// Mitsubishi GX Works2 project: PLC_GROUP21   PLC: FX3G

// global labels: Global1
VAR_GLOBAL
  start_day_switch AT X007 : BOOL;
  start_day_light AT Y007 : BOOL;
  end_day_light AT M3 : BOOL;
  input1 AT D1110 : REAL;
  input2 AT D1120 : REAL;
  input3 AT D1130 : REAL;
  input4 AT D1140 : REAL;
  petel AT D1150 : REAL;
  lemon AT D1160 : REAL;
  stabilizer AT D1170 : REAL;
  gummybears AT D1180 : REAL;
  prepare_switch AT X001 : BOOL;
  regular_gumigam_range AT M20 : BOOL;
  deluxe_gumigam_range AT M19 : BOOL;
END_VAR
VAR_GLOBAL CONSTANT
  const5 : REAL := 5.0;
  const6 : REAL := 6.0;
  divide : REAL := 400.0;
END_VAR
VAR_GLOBAL
  saved_analog AT D7000 : REAL;
  analog_input1 AT D8280 : INT;
END_VAR
VAR_GLOBAL CONSTANT
  min_pete_regular : REAL := 280;
END_VAR
VAR_GLOBAL
  enough_petel_regular AT M60 : BOOL;
END_VAR
VAR_GLOBAL CONSTANT
  min_lemon_regular : REAL := 455;
END_VAR
VAR_GLOBAL
  enough_lemon_regular AT M61 : BOOL;
END_VAR
VAR_GLOBAL CONSTANT
  min_stabilizer_regular : REAL := 105;
END_VAR
VAR_GLOBAL
  enough_gumi_bears AT M63 : BOOL;
END_VAR
VAR_GLOBAL CONSTANT
  min_gummybears_regular : REAL := 28;
END_VAR
VAR_GLOBAL
  enough_stabilizer_regular AT M62 : BOOL;
END_VAR
VAR_GLOBAL CONSTANT
  min_pete_del : REAL := 385;
END_VAR
VAR_GLOBAL
  enough_petel_del AT M50 : BOOL;
END_VAR
VAR_GLOBAL CONSTANT
  min_lemon_del : REAL := 665;
END_VAR
VAR_GLOBAL
  enough_lemon_del AT M51 : BOOL;
END_VAR
VAR_GLOBAL CONSTANT
  min_stabilizer_del : REAL := 210;
END_VAR
VAR_GLOBAL
  enough_stabilizer_del AT M52 : BOOL;
END_VAR
VAR_GLOBAL CONSTANT
  min_gummybears_del : REAL := 70;
END_VAR
VAR_GLOBAL
  enough_gummybears_regular AT M63 : BOOL;
  enough_gummybears_del AT M53 : BOOL;
  help_gate_regular AT M39 : BOOL;
  help_gate_del AT M38 : BOOL;
  enough_in_regularl_stock AT M18 : BOOL;
  enough_in_del_stock AT M40 : BOOL;
  preper_icecream_timer AT TC9 : BOOL;
  const_5 AT K50 : INT;
  preper_icecream_timer_ts9 AT TS9 : BOOL;
  preper_icecream_is_on_light AT Y000 : BOOL;
  preper_is_on_light AT Y000 : BOOL;
END_VAR
VAR_GLOBAL CONSTANT
  time_for_cold_8S : INT := 80;
END_VAR
VAR_GLOBAL
  time_fer AT D1180 : INT;
  sen_10 AT X003 : BOOL;
END_VAR
VAR_GLOBAL CONSTANT
  time_for_fer_const_3S : INT := 3;
  time_for_mix_5S : INT := 50;
  time_for_mix_3S : INT := 30;
END_VAR
VAR_GLOBAL
  Y5_light_on AT Y005 : BOOL;
  Y6_light_on AT Y006 : BOOL;
  Y6_flash_counter AT TC6 : BOOL;
  timer_ts6 AT TS6 : BOOL;
  finish_cold : BOOL;
  packing_switch AT X004 : BOOL;
  counter_pack AT CC3 : BOOL;
  Y4_light_on AT Y004 : BOOL;
  CC3_term AT CS3 : BOOL;
END_VAR
VAR_GLOBAL CONSTANT
  const7 : INT := 7;
  pack_finish : REAL := 1.0;
END_VAR
VAR_GLOBAL
  cont_petel_ice_cream AT D1190 : REAL;
  cont_lemon_ice_cream AT D1200 : REAL;
END_VAR
VAR_GLOBAL CONSTANT
  lemon_for_petel_icecream_regular : REAL := 35;
  stabilizer_for_petel_ice_regular : REAL := 35;
  stabilizer_for_del_icecream : REAL := 140;
  lemon_for_del_icecream : REAL := 560;
  lemon_for_del_lemon_icecream : REAL := 560;
  lemon_for_lemon_icecream_regular : REAL := 420;
  stabilizer_for_lemon_ice_regular : REAL := 70;
  lemon_for_petel_icecream_del : REAL := 105;
  stabilizer_for_petel_ice_del : REAL := 70;
END_VAR
VAR_GLOBAL
  start_cooling AT X002 : BOOL;
  cooling_petel AT D1300 : REAL;
  cooling_lemon AT D1310 : REAL;
END_VAR
VAR_GLOBAL CONSTANT
  stabilizer_for_del_lemon_ice : REAL := 140;
END_VAR
VAR_GLOBAL
  cooling_icecream_timer AT TC8 : BOOL;
  const_8 AT K80 : INT;
  cooling_icecream_timer_ts8 AT TS8 : BOOL;
  cooling_icecream_is_on_light AT Y002 : BOOL;
  stop_cooling AT M10 : BOOL;
END_VAR
VAR_GLOBAL CONSTANT
  update_petel_cont : REAL := 350;
  update_reg_lemon_cont : REAL := 490;
  update_reg_petel_cont : REAL := 350;
  update_del_petel_cont : REAL := 560;
  update_del_lemon_cont : REAL := 700;
END_VAR
VAR_GLOBAL
  mix_cont AT D1320 : REAL;
  time_mix AT D1500 : INT;
  mix_flash_counter AT TC4 : BOOL;
  mix_flash_counter_ts4 AT TS4 : BOOL;
  const_1 AT K10 : INT;
  mix_time_reg AT TC3 : BOOL;
  mix_time_del AT TC5 : BOOL;
END_VAR
VAR_GLOBAL CONSTANT
  const_time_mix_reg : INT := 30;
  const_time_mix_del : INT := 50;
END_VAR
VAR_GLOBAL
  mix_time_reg_ts AT TS3 : BOOL;
  mix_time_del_ts AT TS5 : BOOL;
  start_blinking AT M36 : BOOL;
  Y5_flash_counter AT TC7 : BOOL;
  timer_ts7 AT TS7 : BOOL;
  blink_time AT K10 : INT;
  blinking_help AT M37 : BOOL;
  pack1_switch AT X000 : BOOL;
  count_gumigam_in_box AT CN3 : INT;
END_VAR
VAR_GLOBAL CONSTANT
  no_gumigam : INT;
END_VAR
VAR_GLOBAL
  new_box AT M70 : BOOL;
  end_day_switch AT X005 : BOOL;
  analog_output AT D8282 : INT;
END_VAR
VAR_GLOBAL CONSTANT
  const_40 : REAL := 40;
END_VAR
VAR_GLOBAL
  reg_pack_count_after_mul AT D1404 : REAL;
  input1_petel AT D1110 : REAL;
  input2_lemon AT D1120 : REAL;
  input3_stabilizer AT D1130 : REAL;
  input4_gummybears AT D1140 : REAL;
  pack_total_count AT D1402 : REAL;
  zero AT D5000 : REAL;
  zero_word AT D5010 : INT;
  cont AT D1200 : REAL;
  end_of_iteration AT M80 : BOOL;
  bDIKA AT M90 : BOOL;
END_VAR

// task Task_01 (event TRUE, interval 0, priority 31): POU_01

PROGRAM POU_01
(* structured ladder/FBD written out as ST: instructions are called as NAME(EN, inputs, outputs); _pN, _eN, _tN stand for wires *)
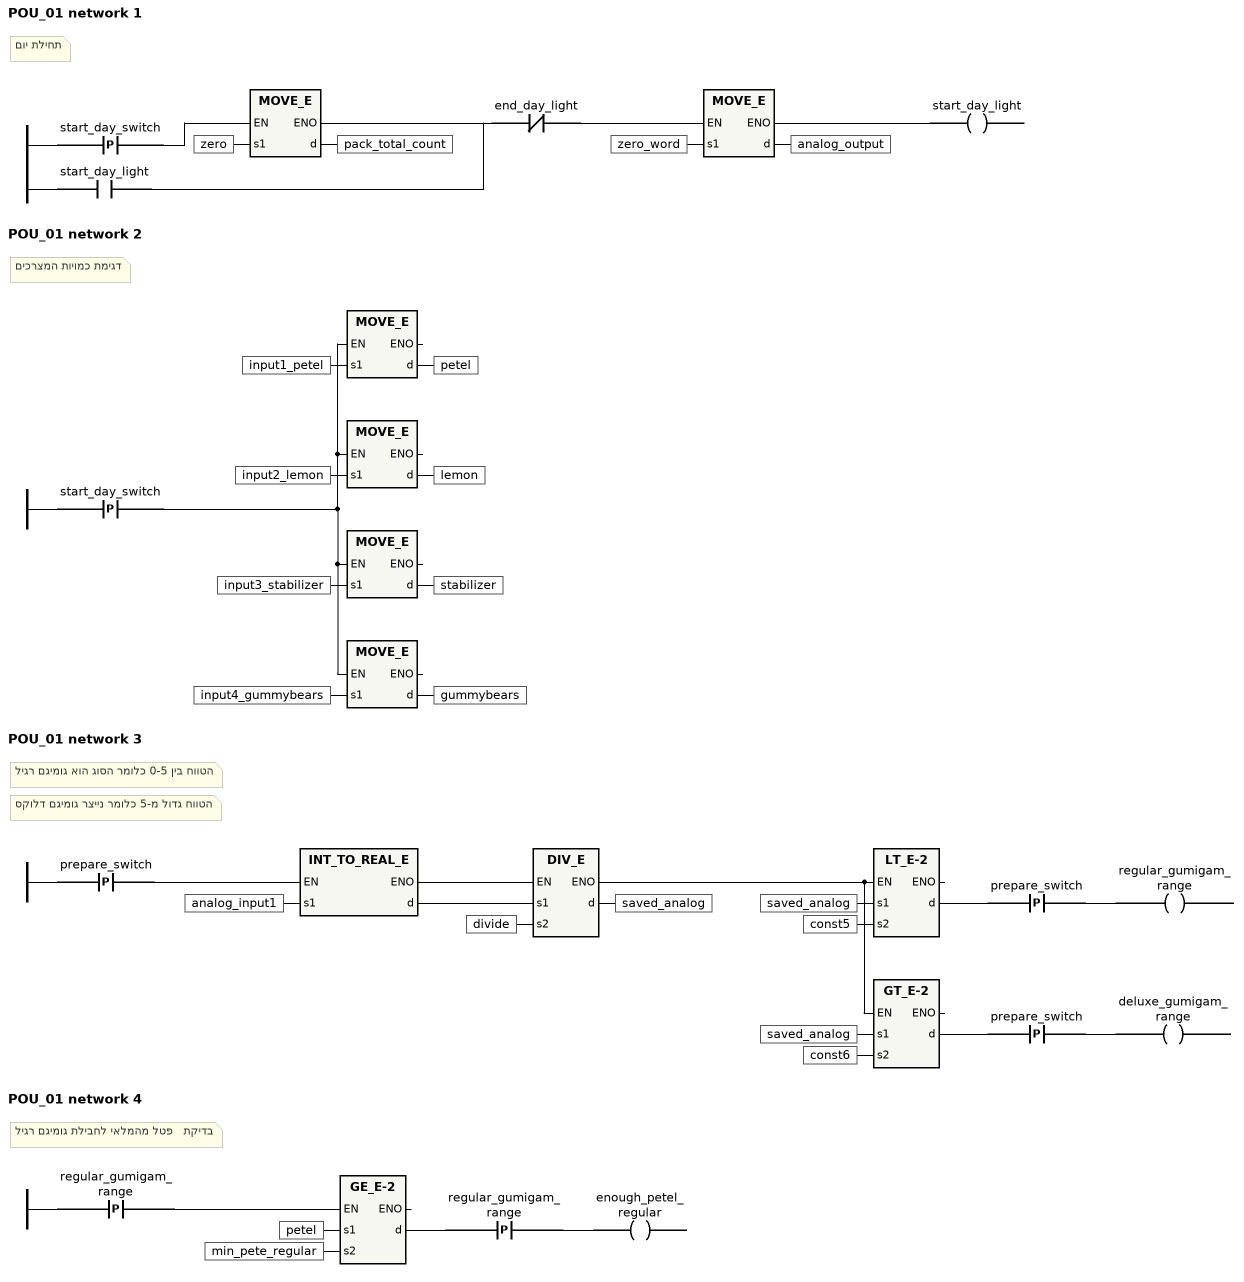
(* network 1 *)
(* תחילת יום *)
_e1 := MOVE_E(LDP(TRUE, start_day_switch), zero, pack_total_count);
_e2 := MOVE_E((_e1 OR start_day_light) AND NOT end_day_light, zero_word, analog_output);
start_day_light := _e2;
(* network 2 *)
(* דגימת כמויות המצרכים *)
_p1 := LDP(TRUE, start_day_switch);
MOVE_E(_p1, input1_petel, petel);
MOVE_E(_p1, input2_lemon, lemon);
MOVE_E(_p1, input3_stabilizer, stabilizer);
MOVE_E(_p1, input4_gummybears, gummybears);
(* network 3 *)
(* הטווח בין 0-5 כלומר הסוג הוא גומיגם רגיל *)
(* הטווח גדול מ-5 כלומר נייצר גומיגם דלוקס *)
_e2 := INT_TO_REAL_E(LDP(TRUE, prepare_switch), analog_input1, _t1);
_e3 := DIV_E(_e2, _t1, divide, saved_analog);
LT_E(_e3, saved_analog, const5, _t4);
regular_gumigam_range := _t4 AND LDP(TRUE, prepare_switch);
GT_E(_e3, saved_analog, const6, _t5);
deluxe_gumigam_range := _t5 AND LDP(TRUE, prepare_switch);
(* network 4 *)
(* בדיקת   פטל מהמלאי לחבילת גומיגם רגיל *)
GE_E(LDP(TRUE, regular_gumigam_range), petel, min_pete_regular, _t1);
enough_petel_regular := _t1 AND LDP(TRUE, regular_gumigam_range);
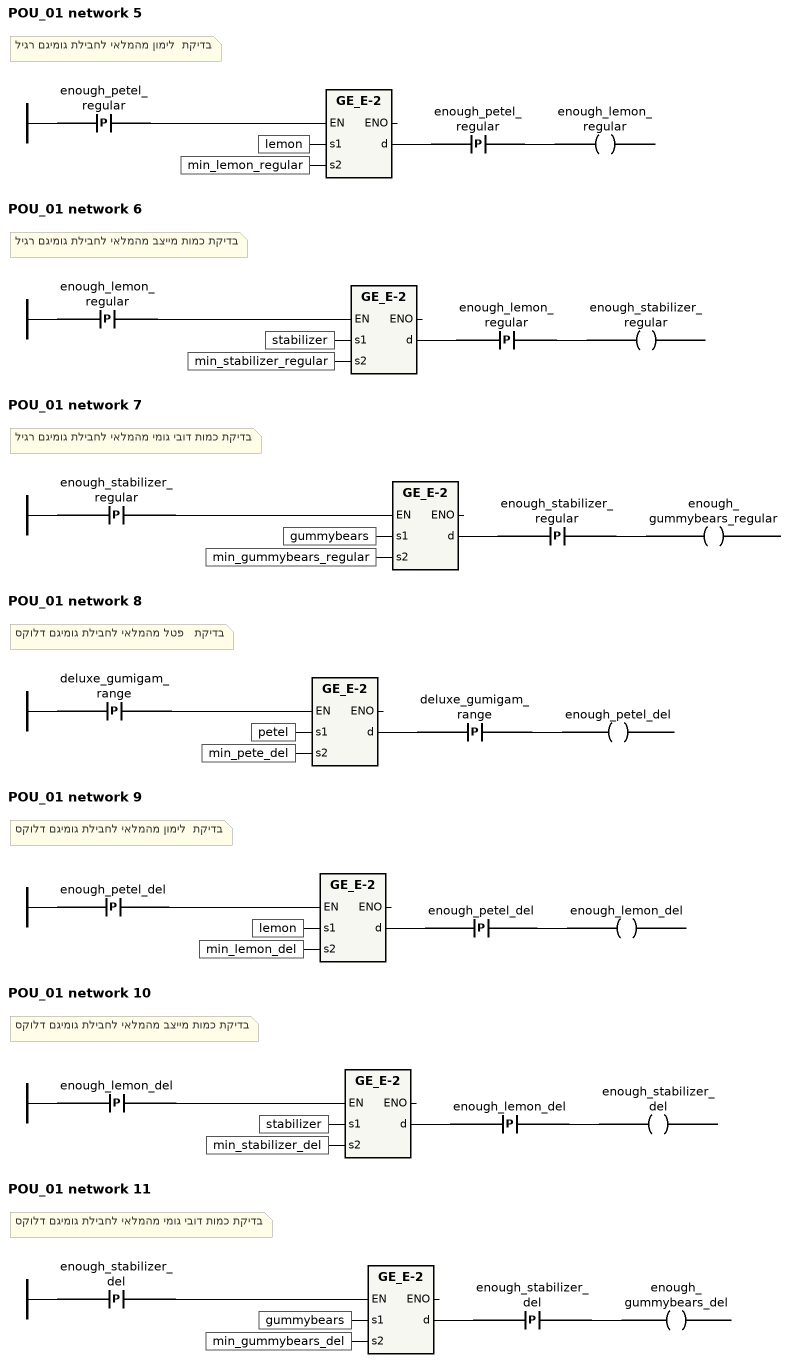
(* network 5 *)
(* בדיקת  לימון מהמלאי לחבילת גומיגם רגיל *)
GE_E(LDP(TRUE, enough_petel_regular), lemon, min_lemon_regular, _t1);
enough_lemon_regular := _t1 AND LDP(TRUE, enough_petel_regular);
(* network 6 *)
(* בדיקת כמות מייצב מהמלאי לחבילת גומיגם רגיל *)
GE_E(LDP(TRUE, enough_lemon_regular), stabilizer, min_stabilizer_regular, _t1);
enough_stabilizer_regular := _t1 AND LDP(TRUE, enough_lemon_regular);
(* network 7 *)
(* בדיקת כמות דובי גומי מהמלאי לחבילת גומיגם רגיל *)
GE_E(LDP(TRUE, enough_stabilizer_regular), gummybears, min_gummybears_regular, _t1);
enough_gummybears_regular := _t1 AND LDP(TRUE, enough_stabilizer_regular);
(* network 8 *)
(* בדיקת   פטל מהמלאי לחבילת גומיגם דלוקס *)
GE_E(LDP(TRUE, deluxe_gumigam_range), petel, min_pete_del, _t1);
enough_petel_del := _t1 AND LDP(TRUE, deluxe_gumigam_range);
(* network 9 *)
(* בדיקת  לימון מהמלאי לחבילת גומיגם דלוקס *)
GE_E(LDP(TRUE, enough_petel_del), lemon, min_lemon_del, _t1);
enough_lemon_del := _t1 AND LDP(TRUE, enough_petel_del);
(* network 10 *)
(* בדיקת כמות מייצב מהמלאי לחבילת גומיגם דלוקס *)
GE_E(LDP(TRUE, enough_lemon_del), stabilizer, min_stabilizer_del, _t1);
enough_stabilizer_del := _t1 AND LDP(TRUE, enough_lemon_del);
(* network 11 *)
(* בדיקת כמות דובי גומי מהמלאי לחבילת גומיגם דלוקס *)
GE_E(LDP(TRUE, enough_stabilizer_del), gummybears, min_gummybears_del, _t1);
enough_gummybears_del := _t1 AND LDP(TRUE, enough_stabilizer_del);
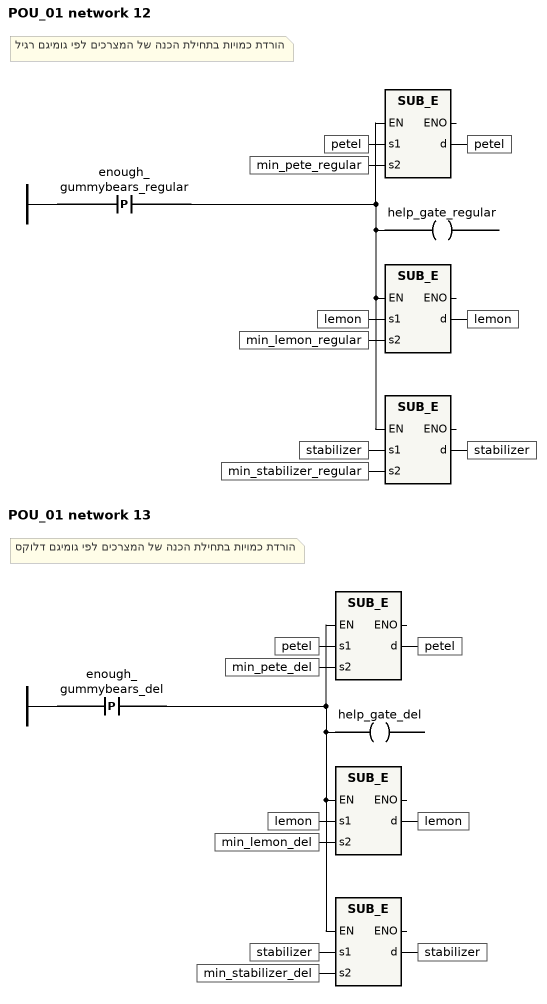
(* network 12 *)
(* הורדת כמויות בתחילת הכנה של המצרכים לפי גומיגם רגיל *)
_p1 := LDP(TRUE, enough_gummybears_regular);
help_gate_regular := _p1;
SUB_E(_p1, petel, min_pete_regular, petel);
SUB_E(_p1, lemon, min_lemon_regular, lemon);
SUB_E(_p1, stabilizer, min_stabilizer_regular, stabilizer);
(* network 13 *)
(* הורדת כמויות בתחילת הכנה של המצרכים לפי גומיגם דלוקס *)
_p1 := LDP(TRUE, enough_gummybears_del);
help_gate_del := _p1;
SUB_E(_p1, petel, min_pete_del, petel);
SUB_E(_p1, lemon, min_lemon_del, lemon);
SUB_E(_p1, stabilizer, min_stabilizer_del, stabilizer);
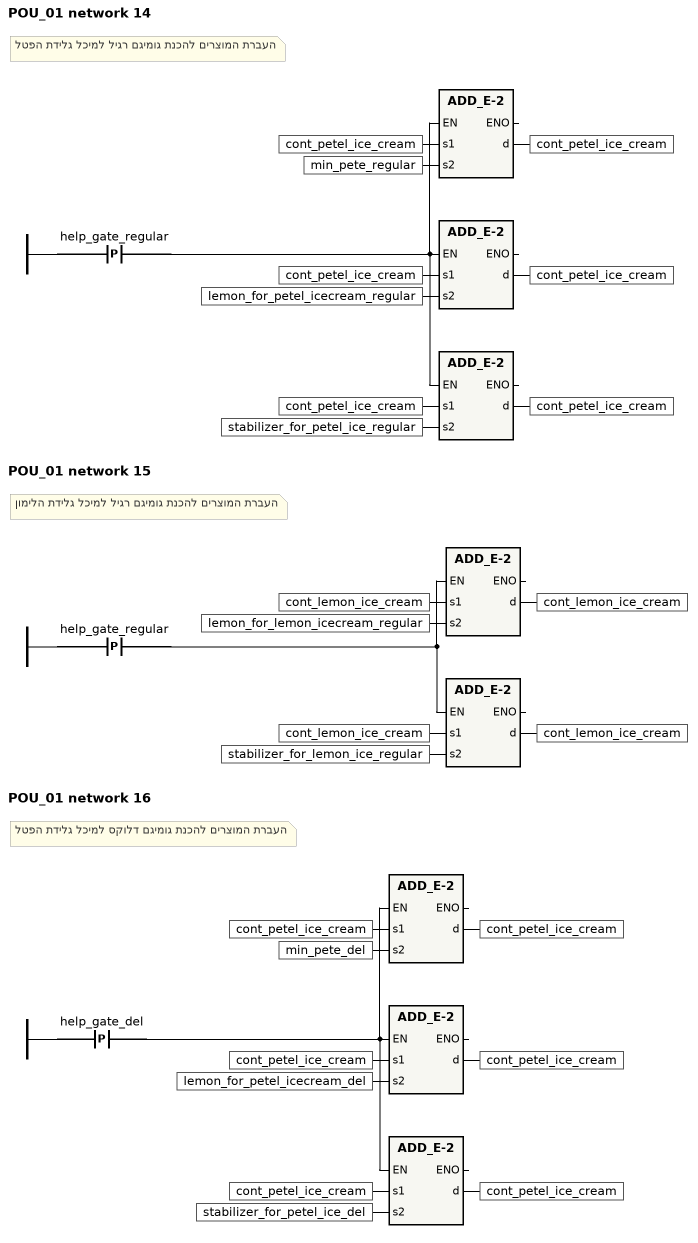
(* network 14 *)
(* העברת המוצרים להכנת גומיגם רגיל למיכל גלידת הפטל *)
_p1 := LDP(TRUE, help_gate_regular);
ADD_E(_p1, cont_petel_ice_cream, min_pete_regular, cont_petel_ice_cream);
ADD_E(_p1, cont_petel_ice_cream, lemon_for_petel_icecream_regular, cont_petel_ice_cream);
ADD_E(_p1, cont_petel_ice_cream, stabilizer_for_petel_ice_regular, cont_petel_ice_cream);
(* network 15 *)
(* העברת המוצרים להכנת גומיגם רגיל למיכל גלידת הלימון *)
_p1 := LDP(TRUE, help_gate_regular);
ADD_E(_p1, cont_lemon_ice_cream, lemon_for_lemon_icecream_regular, cont_lemon_ice_cream);
ADD_E(_p1, cont_lemon_ice_cream, stabilizer_for_lemon_ice_regular, cont_lemon_ice_cream);
(* network 16 *)
(* העברת המוצרים להכנת גומיגם דלוקס למיכל גלידת הפטל *)
_p1 := LDP(TRUE, help_gate_del);
ADD_E(_p1, cont_petel_ice_cream, min_pete_del, cont_petel_ice_cream);
ADD_E(_p1, cont_petel_ice_cream, lemon_for_petel_icecream_del, cont_petel_ice_cream);
ADD_E(_p1, cont_petel_ice_cream, stabilizer_for_petel_ice_del, cont_petel_ice_cream);
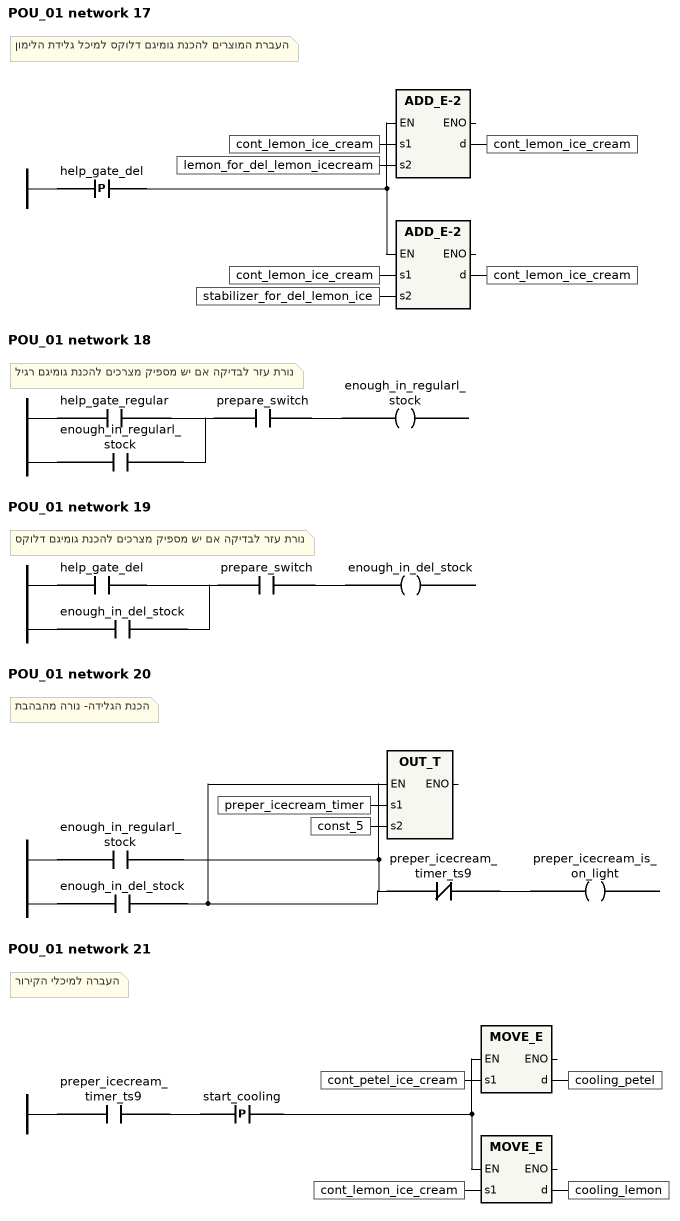
(* network 17 *)
(* העברת המוצרים להכנת גומיגם דלוקס למיכל גלידת הלימון *)
_p1 := LDP(TRUE, help_gate_del);
ADD_E(_p1, cont_lemon_ice_cream, lemon_for_del_lemon_icecream, cont_lemon_ice_cream);
ADD_E(_p1, cont_lemon_ice_cream, stabilizer_for_del_lemon_ice, cont_lemon_ice_cream);
(* network 18 *)
(* נורת עזר לבדיקה אם יש מספיק מצרכים להכנת גומיגם רגיל *)
enough_in_regularl_stock := (help_gate_regular OR enough_in_regularl_stock) AND prepare_switch;
(* network 19 *)
(* נורת עזר לבדיקה אם יש מספיק מצרכים להכנת גומיגם דלוקס *)
enough_in_del_stock := (help_gate_del OR enough_in_del_stock) AND prepare_switch;
(* network 20 *)
(* הכנת הגלידה- נורה מהבהבת *)
_p1 := enough_in_regularl_stock OR enough_in_del_stock;
OUT_T(_p1, preper_icecream_timer, const_5);
preper_icecream_is_on_light := _p1 AND NOT preper_icecream_timer_ts9;
(* network 21 *)
(* העברה למיכלי הקירור *)
_p1 := preper_icecream_timer_ts9 AND LDP(TRUE, start_cooling);
MOVE_E(_p1, cont_petel_ice_cream, cooling_petel);
MOVE_E(_p1, cont_lemon_ice_cream, cooling_lemon);
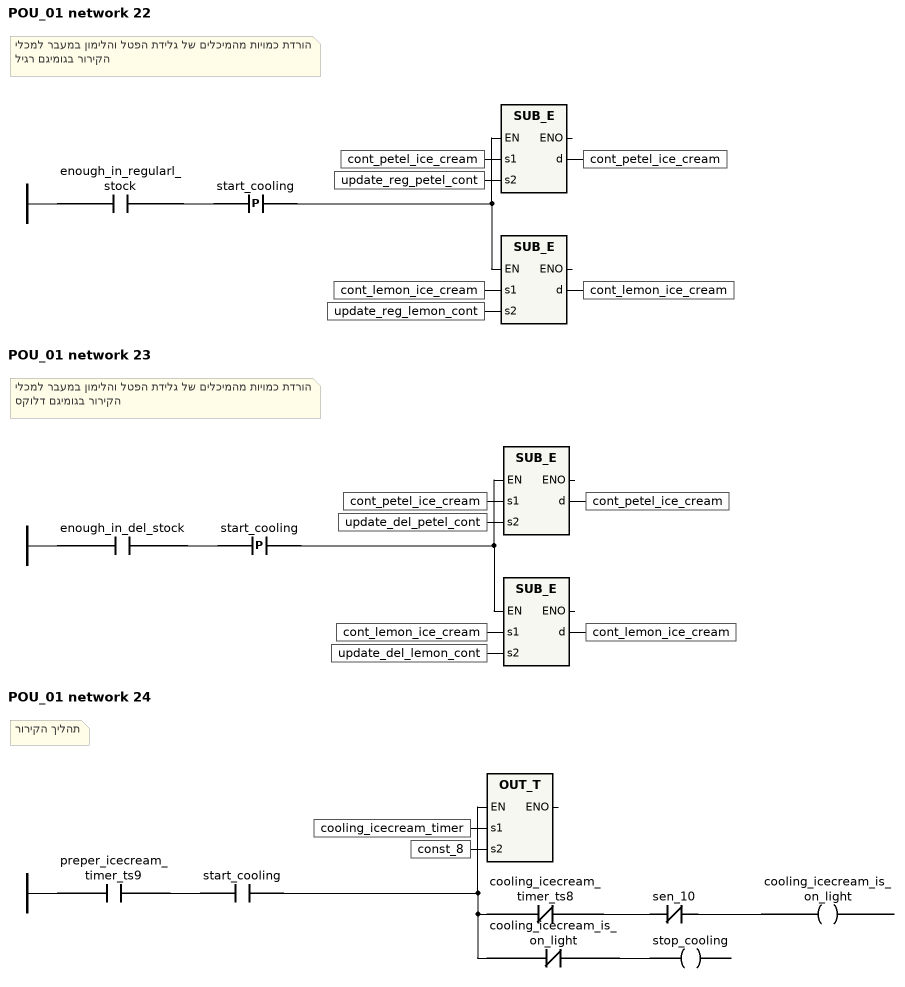
(* network 22 *)
(* הורדת כמויות מהמיכלים של גלידת הפטל והלימון במעבר למכלי הקירור בגומיגם רגיל *)
_p1 := enough_in_regularl_stock AND LDP(TRUE, start_cooling);
SUB_E(_p1, cont_petel_ice_cream, update_reg_petel_cont, cont_petel_ice_cream);
SUB_E(_p1, cont_lemon_ice_cream, update_reg_lemon_cont, cont_lemon_ice_cream);
(* network 23 *)
(* הורדת כמויות מהמיכלים של גלידת הפטל והלימון במעבר למכלי הקירור בגומיגם דלוקס *)
_p1 := enough_in_del_stock AND LDP(TRUE, start_cooling);
SUB_E(_p1, cont_petel_ice_cream, update_del_petel_cont, cont_petel_ice_cream);
SUB_E(_p1, cont_lemon_ice_cream, update_del_lemon_cont, cont_lemon_ice_cream);
(* network 24 *)
(* תהליך הקירור *)
_p1 := preper_icecream_timer_ts9 AND start_cooling;
OUT_T(_p1, cooling_icecream_timer, const_8);
cooling_icecream_is_on_light := _p1 AND NOT cooling_icecream_timer_ts8 AND NOT sen_10;
stop_cooling := _p1 AND NOT cooling_icecream_is_on_light;
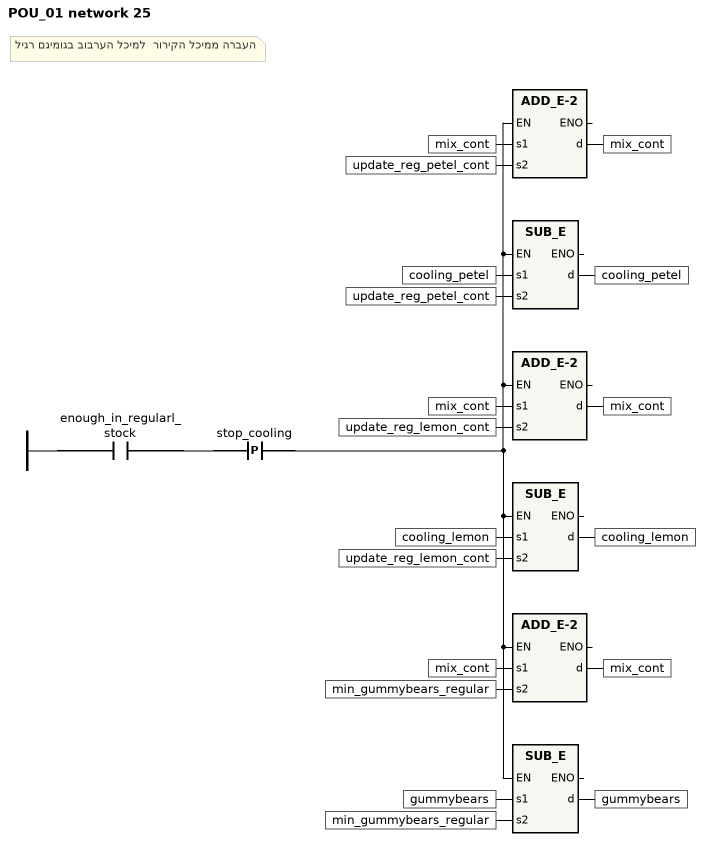
(* network 25 *)
(* העברה ממיכל הקירור  למיכל הערבוב בגומיגם רגיל *)
_p1 := enough_in_regularl_stock AND LDP(TRUE, stop_cooling);
ADD_E(_p1, mix_cont, update_reg_petel_cont, mix_cont);
SUB_E(_p1, cooling_petel, update_reg_petel_cont, cooling_petel);
ADD_E(_p1, mix_cont, update_reg_lemon_cont, mix_cont);
SUB_E(_p1, cooling_lemon, update_reg_lemon_cont, cooling_lemon);
ADD_E(_p1, mix_cont, min_gummybears_regular, mix_cont);
SUB_E(_p1, gummybears, min_gummybears_regular, gummybears);
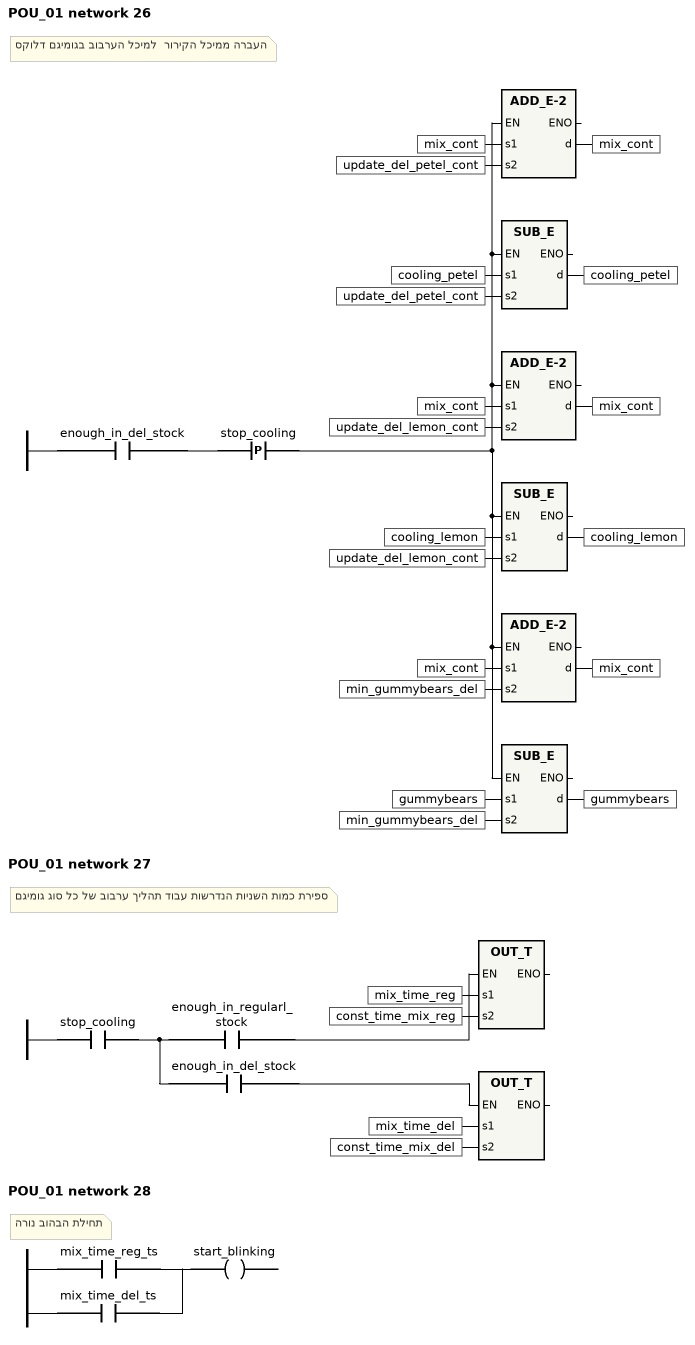
(* network 26 *)
(* העברה ממיכל הקירור  למיכל הערבוב בגומיגם דלוקס *)
_p1 := enough_in_del_stock AND LDP(TRUE, stop_cooling);
ADD_E(_p1, mix_cont, update_del_petel_cont, mix_cont);
SUB_E(_p1, cooling_petel, update_del_petel_cont, cooling_petel);
ADD_E(_p1, mix_cont, update_del_lemon_cont, mix_cont);
SUB_E(_p1, cooling_lemon, update_del_lemon_cont, cooling_lemon);
ADD_E(_p1, mix_cont, min_gummybears_del, mix_cont);
SUB_E(_p1, gummybears, min_gummybears_del, gummybears);
(* network 27 *)
(* ספירת כמות השניות הנדרשות עבוד תהליך ערבוב של כל סוג גומיגם *)
OUT_T(stop_cooling AND enough_in_regularl_stock, mix_time_reg, const_time_mix_reg);
OUT_T(stop_cooling AND enough_in_del_stock, mix_time_del, const_time_mix_del);
(* network 28 *)
(* תחילת הבהוב נורה *)
start_blinking := mix_time_reg_ts OR mix_time_del_ts;
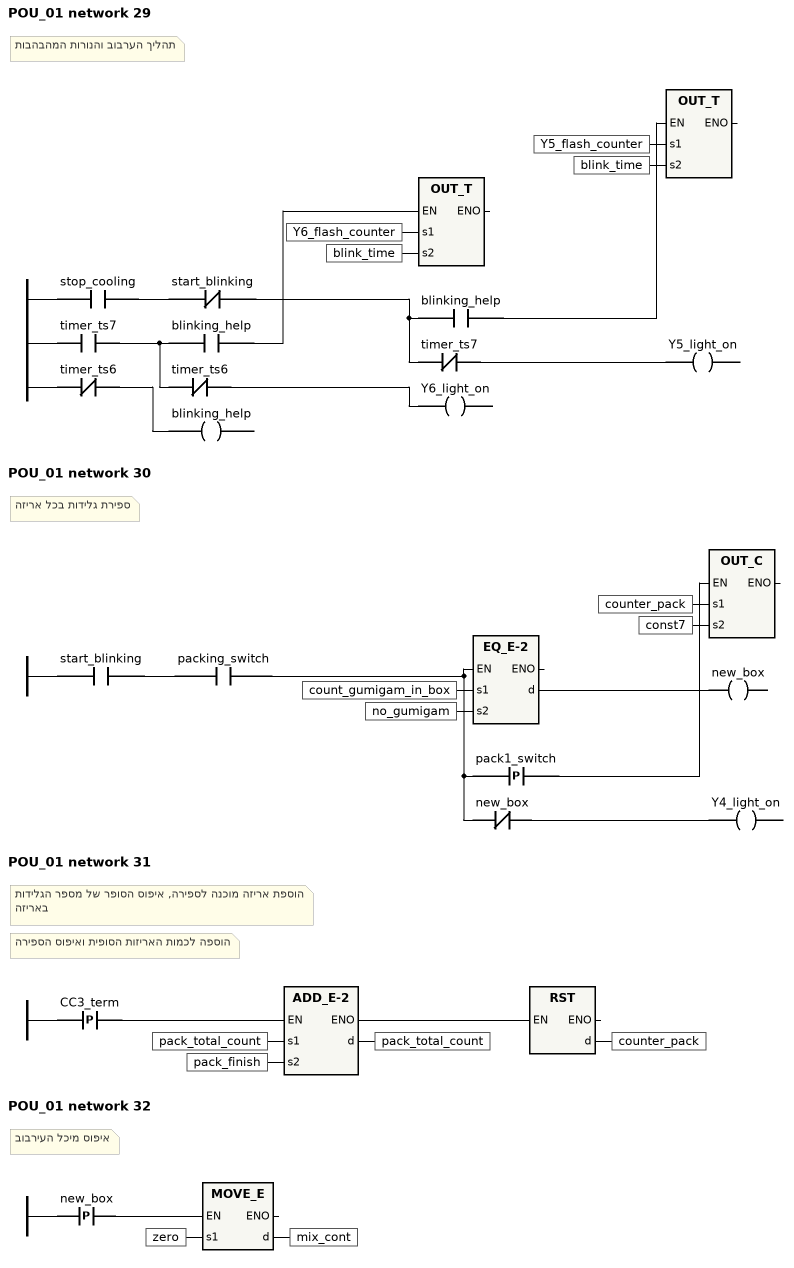
(* network 29 *)
(* תהליך הערבוב והנורות המהבהבות *)
_p1 := stop_cooling AND NOT start_blinking;
OUT_T(_p1 AND blinking_help, Y5_flash_counter, blink_time);
Y5_light_on := _p1 AND NOT timer_ts7;
OUT_T(timer_ts7 AND blinking_help, Y6_flash_counter, blink_time);
Y6_light_on := timer_ts7 AND NOT timer_ts6;
blinking_help := NOT timer_ts6;
(* network 30 *)
(* ספירת גלידות בכל אריזה *)
_p1 := start_blinking AND packing_switch;
OUT_C(_p1 AND LDP(TRUE, pack1_switch), counter_pack, const7);
EQ_E(_p1, count_gumigam_in_box, no_gumigam, _t2);
new_box := _t2;
Y4_light_on := _p1 AND NOT new_box;
(* network 31 *)
(* הוספת אריזה מוכנה לספירה, איפוס הסופר של מספר הגלידות באריזה *)
(* הוספה לכמות האריזות הסופית ואיפוס הספירה *)
_e1 := ADD_E(LDP(TRUE, CC3_term), pack_total_count, pack_finish, pack_total_count);
RST(_e1, counter_pack);
(* network 32 *)
(* איפוס מיכל העירבוב *)
MOVE_E(LDP(TRUE, new_box), zero, mix_cont);
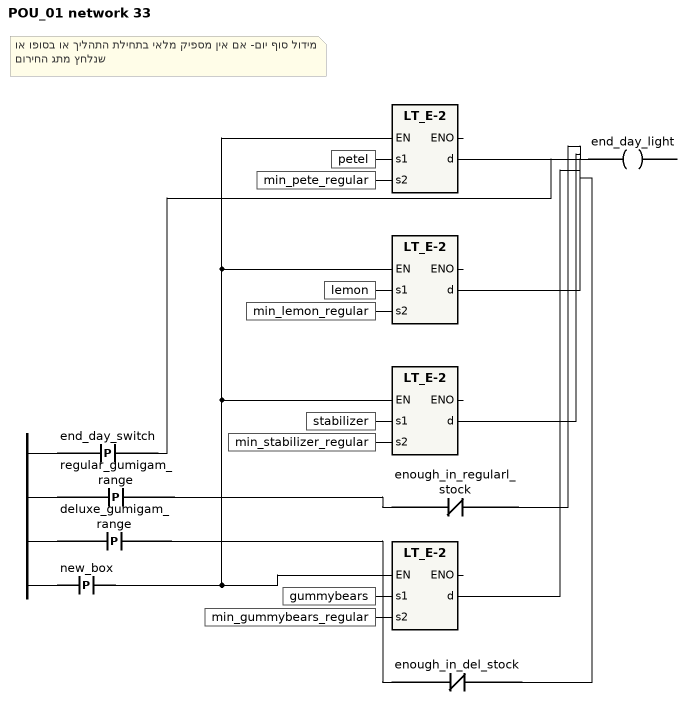
(* network 33 *)
(* מידול סוף יום- אם אין מספיק מלאי בתחילת התהליך או בסופו או שנלחץ מתג החירום *)
_p1 := LDP(TRUE, new_box);
LT_E(_p1, petel, min_pete_regular, _t2);
LT_E(_p1, lemon, min_lemon_regular, _t3);
LT_E(_p1, stabilizer, min_stabilizer_regular, _t4);
LT_E(_p1, gummybears, min_gummybears_regular, _t5);
end_day_light := LDP(TRUE, end_day_switch) OR (LDP(TRUE, regular_gumigam_range) AND NOT enough_in_regularl_stock) OR (LDP(TRUE, deluxe_gumigam_range) AND NOT enough_in_del_stock) OR _t2 OR _t3 OR _t4 OR _t5;
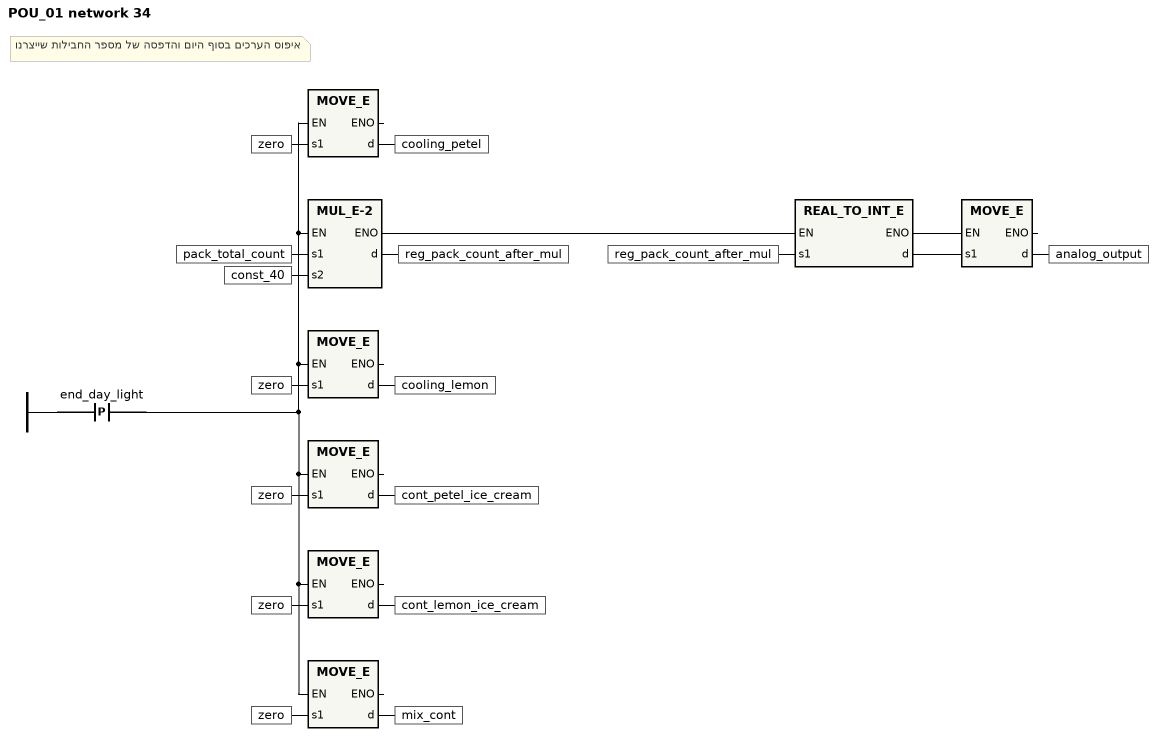
(* network 34 *)
(* איפוס הערכים בסוף היום והדפסה של מספר החבילות שייצרנו *)
_p1 := LDP(TRUE, end_day_light);
MOVE_E(_p1, zero, cooling_petel);
MOVE_E(_p1, zero, cooling_lemon);
MOVE_E(_p1, zero, cont_petel_ice_cream);
MOVE_E(_p1, zero, cont_lemon_ice_cream);
MOVE_E(_p1, zero, mix_cont);
_e2 := MUL_E(_p1, pack_total_count, const_40, reg_pack_count_after_mul);
_e4 := REAL_TO_INT_E(_e2, reg_pack_count_after_mul, _t3);
MOVE_E(_e4, _t3, analog_output);
END_PROGRAM
